(* CODESYS project verseny2

Project tree, tasks and I/O mapping:
  Device : CODESYS Control for PFC200 SL, 3S - Smart Software Solutions GmbH, version 4.1.0.0
    application Application
      libraries: Standard, * (System)
      task MainTask (cyclic, interval t#20ms, priority 1) calls MANUAL_TEST, input_led
      Andris/
        program prg_Beolvasas [ST]
        program prgBeolvasas_Sagaval_kezdunk [ST]
        program prgBeolvasas_Zoldel_kezdunk [ST]
      enum/
        data type enuIranyok
        data type enuMain
        data type enuSzinek
      data type enumRobotok
      fb/
        function block fbBLINKER2 [ST]
        function block fbBLINKER4 [ST]
        function block fbKombi3 [ST]
        function block fbKombi4 [ST]
      fun/
        function funAGV1_Location [ST]
        function funAGV2_Location [ST]
        function funAVG1_Set_Destination_1 [ST]
        function funAVG1_Set_Destination [ST]
        function funSargaElsoOszlopCheck [ST]
        function funTombfordito [ST]
        function funTombMaximuma [ST]
        function funTombMinimuma [ST]
        function funTombRendezesBuborek [ST]
        function funZoldElsoOszlopCheck [ST]
      global variables GVL
      global variables I
      program input_led [ST]
      Magocsi/
        function block fbMozgatas_zold [ST]
        function block fbRendezes [ST]
        function block fbRobotMozgas [ST]
      program MANUAL_TEST [ST]
      program PLC_PRG [ST]
      prg/
        program prgTEST1 [ST]
        program prgTEST2 [ST]
      global variables Q
      Ricsi/
        program prgEllenorzes [ST]
        program prgEmel [ST]
        program prgLerak [ST]
        program prgRaktar_sor1_bol_vegpontba [ST]
        program prgRaktarazas [ST]
        program prgSarga [ST]
        program prgZold [ST]
        program TEST [ST]
      program state_machine_main [ST]
    Pfc200Bus : Wago PFC200 internal bus, 3S - Smart Software Solutions GmbH, version 4.1.0.0
      _750_14xx : 16DI, WAGO Kontakttechnik GmbH u. Co. KG, order no. 750-14xx, version 4.1.0.0
          unmapped channels: %IW5 Digital Inputs 0 - 15
      _750_14xx_1 : 16DI, WAGO Kontakttechnik GmbH u. Co. KG, order no. 750-14xx, version 4.1.0.0
          unmapped channels: %IW20 Digital Inputs 0 - 15
      _750_15xx_1 : 16DO, WAGO Kontakttechnik GmbH u. Co. KG, order no. 750-15xx, version 4.1.0.0
          unmapped channels: %QW20 Digital Outputs 0 - 15
      _750_15xx : 16DO, WAGO Kontakttechnik GmbH u. Co. KG, order no. 750-15xx, version 4.1.0.0
          unmapped channels: %QW5 Digital Outputs 0 - 15
      _75x_459 : 75x-459/0..-000 4AI, 0-10 V, WAGO Kontakttechnik GmbH u. Co. KG, order no. 75x-459(/0..-000), version 4.1.0.0
          unmapped channels: Analog Input Channel 0, Analog Input Channel 1, Analog Input Channel 2, Analog Input Channel 3
      _75x_559 : 75x-559/0..-000 4AO, 0-10 V, WAGO Kontakttechnik GmbH u. Co. KG, order no. 75x-559(/0..-000), version 4.1.0.0
          unmapped channels: Analog Output Channel 0, Analog Output Channel 1, Analog Output Channel 2, Analog Output Channel 3
*)

// Device/Application/enumRobotok
{attribute 'qualified_only'}
{attribute 'strict'}
TYPE enumRobotok :
(
	AGV_Sarga,
	AGV_Zold
);
END_TYPE

// Device/Application/enum/enuIranyok
{attribute 'qualified_only'}
{attribute 'strict'}
TYPE enuIranyok :
(
	felfele,
	lefele,
	balra,
	jobbra
);
END_TYPE

// Device/Application/enum/enuMain
{attribute 'qualified_only'}
{attribute 'strict'}
TYPE enuMain :
(
	wait,
	init,
	beolvasas,
	rendezes,
	done
	
) := wait;
END_TYPE

// Device/Application/enum/enuSzinek
{attribute 'qualified_only'}
{attribute 'strict'}
TYPE enuSzinek :
(
	empty,
	zold,
	sarga,
	kek
);
END_TYPE

// Device/Application/GVL
{attribute 'qualified_only'}
VAR_GLOBAL
	start_r_trig: R_TRIG;
	start_f_trig: F_TRIG;
	stop_r_trig: R_TRIG;
	stop_f_trig: F_TRIG;
	emerg_r_trig: R_TRIG;
	emerg_f_trig: F_TRIG;
	
	aiTombSzinek: ARRAY [0..15] OF INT := [0,-1,-1,-1,-1,-1,-1,-1,-1,-1,0,0,0,0,0,0];
	axTombRobot1Zold: ARRAY [0..15] OF BOOL := [16(TRUE)];
	axTombRobot2Sarga: ARRAY [0..15] OF BOOL := [16(TRUE)];
END_VAR

// Device/Application/I
{attribute 'qualified_only'}
VAR_GLOBAL
	TEST0 AT %IX10.0 : BOOL;
	TEST1 AT %IX10.1 : BOOL;
	TEST2 AT %IX10.2 : BOOL;
	TEST3 AT %IX10.3 : BOOL;
	TEST4 AT %IX10.4 : BOOL;
	TEST5 AT %IX10.5 : BOOL;
	TEST6 AT %IX10.6 : BOOL;
	TEST7 AT %IX10.7 : BOOL;
	TEST8 AT %IX11.0 : BOOL;
	TEST9 AT %IX11.1 : BOOL;
	TEST10 AT %IX11.2 : BOOL;
	TEST11 AT %IX11.3 : BOOL;
	TEST12 AT %IX11.4 : BOOL;
	TEST13 AT %IX11.5 : BOOL;
	TEST14 AT %IX11.6 : BOOL;
	TEST15 AT %IX11.7 : BOOL;
	
	i0 AT %IX40.0 : BOOL;
	i1 AT %IX40.1 : BOOL;
	i2 AT %IX40.2 : BOOL;
	i3 AT %IX40.3 : BOOL;
	i4 AT %IX40.4 : BOOL;
	i5 AT %IX40.5 : BOOL;
	i6 AT %IX40.6 : BOOL;
	i7 AT %IX40.7 : BOOL;
	i8 AT %IX41.0 : BOOL;
	i9 AT %IX41.1 : BOOL;
	i10 AT %IX41.2 : BOOL;
	i11 AT %IX41.3 : BOOL;
	i12 AT %IX41.4 : BOOL;
	i13 AT %IX41.5 : BOOL;
	i14 AT %IX41.6 : BOOL;
	i15 AT %IX41.7 : BOOL;
END_VAR

// Device/Application/Q
{attribute 'qualified_only'}
VAR_GLOBAL
	TEST0 AT %QX10.0 : BOOL;
	TEST1 AT %QX10.1 : BOOL;
	TEST2 AT %QX10.2 : BOOL;
	TEST3 AT %QX10.3 : BOOL;
	TEST4 AT %QX10.4 : BOOL;
	TEST5 AT %QX10.5 : BOOL;
	TEST6 AT %QX10.6 : BOOL;
	TEST7 AT %QX10.7 : BOOL;
	TEST8 AT %QX11.0 : BOOL;
	TEST9 AT %QX11.1 : BOOL;
	TEST10 AT %QX11.2 : BOOL;
	TEST11 AT %QX11.3 : BOOL;
	TEST12 AT %QX11.4 : BOOL;
	TEST13 AT %QX11.5 : BOOL;
	TEST14 AT %QX11.6 : BOOL;
	TEST15 AT %QX11.7 : BOOL;
	
	q0 AT %QX40.0 : BOOL;
	q1 AT %QX40.1 : BOOL;
	q2 AT %QX40.2 : BOOL;
	q3 AT %QX40.3 : BOOL;
	q4 AT %QX40.4 : BOOL;
	q5 AT %QX40.5 : BOOL;
	q6 AT %QX40.6 : BOOL;
	q7 AT %QX40.7 : BOOL;
	q8 AT %QX41.0 : BOOL;
	q9 AT %QX41.1 : BOOL;
	q10 AT %QX41.2 : BOOL;
	q11 AT %QX41.3 : BOOL;
	q12 AT %QX41.4 : BOOL;
	q13 AT %QX41.5 : BOOL;
	q14 AT %QX41.6 : BOOL;
	q15 AT %QX41.7 : BOOL;
	

	
END_VAR

// Device/Application/MANUAL_TEST
PROGRAM MANUAL_TEST
VAR
END_VAR

//KONZOL MUKODTETI AZ OUTPUTOKAT
%QW20:= %IW5;

END_PROGRAM

// Device/Application/input_led
PROGRAM input_led
VAR
END_VAR

//INPUT A KONZOL LEDEKEN
%QW5:= %IW20;

END_PROGRAM

// Device/Application/PLC_PRG
PROGRAM PLC_PRG
VAR
END_VAR

END_PROGRAM

// Device/Application/state_machine_main
PROGRAM state_machine_main
VAR
	iState : enuMain;
	mem_robot : enumRobotok;
END_VAR

CASE iState OF
enuMain.wait:
	
	IF ( ( i.AGV1_L0 OR i.AGV1_L1 OR i.AGV1_L2 OR i.AGV1_L3 ) AND 
		(i.AGV2_L0 OR i.AGV2_L1 OR i.AGV2_L2 OR i.AGV2_L3)) THEN
		iState := enuMain.init;
	END_IF

enuMain.init:
	gvl.axTombRobot1Zold[funAGV1_Location()] := FALSE;
	gvl.axTombRobot2Sarga[funAGV2_Location()] := FALSE;
	IF gvl.axTombRobot1Zold[10] = FALSE THEN
		mem_robot := enumRobotok.AGV_Zold;
	ELSE
		mem_robot := enumRobotok.AGV_Sarga;
	END_IF
	
	iState := enuMain.beolvasas;	
enuMain.beolvasas:
	IF mem_robot = enumRobotok.AGV_Zold THEN
		prgBeolvasas_Zoldel_kezdunk();
	ELSE
		prgBeolvasas_Sagaval_kezdunk();
	END_IF
	
	IF prgBeolvasas_Sagaval_kezdunk.xDone OR prgBeolvasas_Zoldel_kezdunk.xDone THEN
		iState := enuMain.rendezes;
	END_IF 

	
enuMain.rendezes:
enuMain.done:	
END_CASE

END_PROGRAM

// Device/Application/fun/funAGV1_Location
FUNCTION funAGV1_Location : int
VAR_INPUT
END_VAR
VAR
END_VAR

funAGV1_Location := (TO_INT(i.AGV1_L0)) * 1 + (TO_INT(i.AGV1_L1)) * 2 
+ (TO_INT(i.AGV1_L2)) * 4 +(TO_INT( i.AGV1_L3)) * 8;
RETURN;

END_FUNCTION

// Device/Application/fun/funAGV2_Location
FUNCTION funAGV2_Location : int
VAR_INPUT
END_VAR
VAR
END_VAR

funAGV2_Location := i.AGV2_L0 * 1 + i.AGV2_L1 * 2 + i.AGV2_L2 * 4 + i.AGV2_L3 * 8;
RETURN;

END_FUNCTION

// Device/Application/Andris/prgBeolvasas_Zoldel_kezdunk
PROGRAM prgBeolvasas_Zoldel_kezdunk
VAR
	state_Zold : INT;
	state_Sarga : INT;
	lepesek_zold : INT;
	index1 : INT := 4;
	index2 : INT := 5;
	
	fbZold : fbRobotMozgas;
	fbSarga : fbRobotMozgas;
	
END_VAR

VAR_OUTPUT
	xDone : BOOL;
END_VAR

CASE state_Zold OF
// ZOLD MOZGATAS
0:
//10 - > 1
	fbZold(xEnable := TRUE , melyik_mozog := enumRobotok.AGV_Zold , merre_mozog := 1);
	IF fbZold.xDone THEN
		state_Zold := 1;
		gvl.aiTombSzinek[1] := TO_INT(i.AGV1_ID0)*1 + TO_INT(i.AGV1_ID1)*2;
	END_IF
1:
//1 - > 4 -> 7 -> 2
WHILE index1 > -1  DO
	fbZold(xEnable := TRUE , melyik_mozog := enumRobotok.AGV_Zold , merre_mozog := index1);
	
	IF fbZold.xDone THEN
	gvl.aiTombSzinek[index1] := TO_INT(i.AGV1_ID0)*1 + TO_INT(i.AGV1_ID1)*2;
		IF index1 = 7 THEN
			index1 := 8;	
		ELSE
			IF lepesek_zold <= 3 THEN
				index1 := index1 + 3;
			ELSE
				index1 := index1 - 3;
			END_IF
		END_IF
	lepesek_zold := lepesek_zold + 1;
	
	END_IF
	
END_WHILE

IF index1 < 0  THEN
	state_Zold := 3;
END_IF
3:
// DONE
END_CASE


CASE state_Sarga OF

0:
//15 -> 10
	fbSarga(xEnable := TRUE , merre_mozog := 10 , melyik_mozog := enumRobotok.AGV_Sarga );
	IF fbSarga.xDone THEN
		state_Sarga := 1;
	END_IF
1:
//10 -> 3	
	fbSarga(xEnable := TRUE , merre_mozog := 3 , melyik_mozog := enumRobotok.AGV_Sarga );
	IF fbSarga.xDone THEN
		state_Sarga := 2;
		gvl.aiTombSzinek[3] := TO_INT(i.AGV2_ID0)*1 + TO_INT(i.AGV2_ID1)*2;
	END_IF
2:
//3 -> 9
	WHILE index2 < 10  DO
		fbSarga(xEnable := TRUE , merre_mozog := index2 , melyik_mozog := enumRobotok.AGV_Sarga );
		IF fbSarga.xDone THEN
			gvl.aiTombSzinek[index2] := TO_INT(i.AGV2_ID0)*1 + TO_INT(i.AGV2_ID1)*2;
			index2 := index2 +3;
		END_IF

	END_WHILE
	
	IF index2 > 9 THEN
		state_Sarga := 3;
	END_IF
3:
//DONE
END_CASE

IF (state_Sarga = 3) AND (state_Zold = 3) THEN
	xDone := TRUE;
END_IF

END_PROGRAM

// Device/Application/Magocsi/fbRobotMozgas
FUNCTION_BLOCK fbRobotMozgas
VAR_INPUT
	melyik_mozog: INT;
	merre_mozog: INT;
	xEnable: BOOL;
END_VAR
VAR_OUTPUT
	xDone: BOOL;
END_VAR
VAR
	iStateRobotMozgas: INT;
END_VAR

IF NOT xEnable THEN
	RETURN;
END_IF

CASE melyik_mozog OF
	//zold robot
	enumRobotok.AGV_Zold:
		CASE iStateRobotMozgas OF
			0: 
				xDone := FALSE;
				
				funAVG1_Set_Destination(merre_mozog);
				q.AGV1_START := TRUE;
				
				iStateRobotMozgas := 1;
				
			1:
				IF funAGV1_Location() = 0 THEN
					q.AGV1_START := FALSE;
					
					iStateRobotMozgas := 2;
				END_IF
				
			2:
				IF funAgv1_location() > 0 THEN
					iStateRobotMozgas := 0;
					xDone := TRUE;
				END_IF
		END_CASE
		
	//sarga robot
	enumRobotok.AGV_Sarga:
		CASE iStateRobotMozgas OF
			0: 
				xDone := FALSE;
				
				funAVG2_Set_Destination(merre_mozog);
				q.AGV2_START := TRUE;
				
				iStateRobotMozgas := 1;
				
			1:
				IF funAGV2_Location() = 0 THEN
					q.AGV2_START := FALSE;
					
					iStateRobotMozgas := 2;
				END_IF
				
			2:
				IF funAgv2_location() > 0 THEN
					iStateRobotMozgas := 0;
					xDone := TRUE;
				END_IF
		END_CASE
END_CASE

END_FUNCTION_BLOCK

// Device/Application/fun/funAVG1_Set_Destination
FUNCTION funAVG1_Set_Destination : int
VAR_INPUT
	index : INT;
END_VAR
VAR
END_VAR

q.AGV1_D0 := index.0;
q.AGV1_D1 := index.1;
q.AGV1_D2 := index.2;
q.AGV1_D3 := index.3;

END_FUNCTION

// Device/Application/Andris/prgBeolvasas_Sagaval_kezdunk
PROGRAM prgBeolvasas_Sagaval_kezdunk
VAR
	state_Zold : INT;
	state_Sarga : INT;
	lepesek_zold : INT;
	lepesek_sarga : INT ;
	index1 : INT := 4;
	index2 : INT := 5;
	
	fbZold : fbRobotMozgas;
	fbSarga : fbRobotMozgas;
	
END_VAR

VAR_OUTPUT
	xDone : BOOL;
END_VAR

CASE state_Sarga OF
// Sarga MOZGATAS
0:
//10 - > 1
	fbSarga(xEnable := TRUE , melyik_mozog := enumRobotok.AGV_Sarga , merre_mozog := 1);
	IF fbSarga.xDone THEN
		state_Sarga := 1;
		gvl.aiTombSzinek[1] := TO_INT(i.AGV1_ID0)*1 + TO_INT(i.AGV1_ID1)*2;
	END_IF
1:
//1 - > 4 -> 7 -> 2
WHILE index1 > -1  DO
	fbSarga(xEnable := TRUE , melyik_mozog := enumRobotok.AGV_Sarga , merre_mozog := index1);
	
	IF fbSarga.xDone THEN
	gvl.aiTombSzinek[index1] := TO_INT(i.AGV1_ID0)*1 + TO_INT(i.AGV1_ID1)*2;
		IF index1 = 7 THEN
			index1 := 8;	
		ELSE
			IF lepesek_Sarga <= 3 THEN
				index1 := index1 + 3;
			ELSE
				index1 := index1 - 3;
			END_IF
		END_IF
	lepesek_Sarga := lepesek_Sarga + 1;
	
	END_IF
	
END_WHILE

IF index1 < 0  THEN
	state_Sarga := 3;
END_IF
3:
// DONE
END_CASE


CASE state_Zold OF

0:
//15 -> 10
	fbZold(xEnable := TRUE , merre_mozog := 10 , melyik_mozog := enumRobotok.AGV_Zold );
	IF fbZold.xDone THEN
		state_Zold := 1;
	END_IF
1:
//10 -> 3	
	fbZold(xEnable := TRUE , merre_mozog := 3 , melyik_mozog := enumRobotok.AGV_Zold );
	IF fbZold.xDone THEN
		state_Zold := 2;
		gvl.aiTombSzinek[3] := TO_INT(i.AGV2_ID0)*1 + TO_INT(i.AGV2_ID1)*2;
	END_IF
2:
//3 -> 9
	WHILE index2 < 10  DO
		fbZold(xEnable := TRUE , merre_mozog := index2 , melyik_mozog := enumRobotok.AGV_Zold );
		IF fbZold.xDone THEN
			gvl.aiTombSzinek[index2] := TO_INT(i.AGV2_ID0)*1 + TO_INT(i.AGV2_ID1)*2;
			index2 := index2 +3;
		END_IF

	END_WHILE
	
	IF index2 > 9 THEN
		state_Zold := 3;
	END_IF
3:
//DONE
END_CASE

IF (state_Sarga = 3) AND (state_Zold = 3) THEN
	xDone := TRUE;
END_IF

END_PROGRAM

// Device/Application/Andris/prg_Beolvasas
PROGRAM prg_Beolvasas
VAR
	state_Zold : INT;
	state_Sarga : INT;
	fbZold : fbRobotMozgas;
	fbSarga : fbRobotMozgas;
	index1 : INT := 4;
END_VAR

VAR_OUTPUT
	xDone : BOOL;
END_VAR

VAR_INPUT 
	Melyik_van_a_10_en : enumRobotok;
END_VAR

IF Melyik_van_a_10_en = enumRobotok.AGV_Zold THEN

CASE state_Zold OF
// ZOLD MOZGATAS
0:
//10 - > 1
	fbZold(xEnable := TRUE , melyik_mozog := enumRobotok.AGV_Zold , merre_mozog := 1);
	IF fbZold.xDone THEN
		state_Zold := 2;
	END_IF
2:
//1 - > 4 -> 7 -> 2
WHILE NOT (index1 = 2) DO
	
END_WHILE

3:
/

END_CASE

ELSE
	
END_IF

END_PROGRAM

// Device/Application/fb/fbBLINKER2
(*
EZ A FUNKCIO BLOK EGY VILLOGOT VALOSIT MEG AMINEK MINT 
A BEKAPCSOLT IDEJÉT MINT A KIKAPCSOLT IDEJÉT TUDJUK ÁLLITANI.
*)
FUNCTION_BLOCK fbBLINKER2 
VAR_INPUT
	ENABLE : BOOL;
	TIME_ON : TIME ;
	TIME_OFF : TIME;
END_VAR
VAR_OUTPUT
	Q : BOOL;
END_VAR
VAR
	TIMER1 : TON;
	TIMER2 : TON;
	state : INT := 0;
END_VAR

IF ENABLE THEN

TIMER1(IN := state = 0,PT := TIME_ON);
TIMER2(IN := state = 1  , PT := TIME_OFF);

CASE state OF
0:
// ON 
	Q := TRUE;
	IF timer1.Q THEN
		state := 1;
	END_IF
1:
// OFF
	Q := FALSE;
	IF timer2.Q THEN
		state := 0;
	END_IF
	
END_CASE
ELSE
	q := false;
END_IF

END_FUNCTION_BLOCK

// Device/Application/fb/fbBLINKER4
(*
EZ A FUNKCIO BLOK EGY DUPLA VILLOGOT VALOSIT MEG AMINEK MINT 
A BEKAPCSOLT IDEJÉT MINT A KIKAPCSOLT IDEJÉT TUDJUK ÁLLITANI.
*)
FUNCTION_BLOCK fbBLINKER4 
VAR_INPUT
	ENABLE : BOOL;
	TIME_ON1 : TIME ;
	TIME_OFF1 : TIME;
	TIME_ON2 : TIME ;
	TIME_OFF2 : TIME;
END_VAR
VAR_OUTPUT
	Q : BOOL;
END_VAR
VAR
	TIMER0 : TON;
	TIMER1 : TON;
	TIMER2 : TON;
	TIMER3 : TON;
	state : INT := 0;
END_VAR

IF ENABLE THEN

TIMER0(IN := state = 0  , PT := TIME_ON1);
TIMER1(IN := state = 1  , PT := TIME_OFF1);
TIMER2(IN := state = 2  , PT := TIME_ON2);
TIMER3(IN := state = 3  , PT := TIME_OFF2);

CASE state OF
0:
// ON1
	Q := TRUE;
	IF timer0.Q THEN
		state := 1;
	END_IF
1:
// OFF1
	Q := FALSE;
	IF timer1.Q THEN
		state := 2;
	END_IF
2:
// ON2
	Q := TRUE;
	IF timer2.Q THEN
		state := 3;
	END_IF
3:
// OFF2
	Q := FALSE;
	IF timer3.Q THEN
		state := 0;
	END_IF
	
END_CASE
ELSE
	q := FALSE ;
END_IF

END_FUNCTION_BLOCK

// Device/Application/fb/fbKombi3
(*
EZ A FUNKCIO BLOK EGY 3 BEMENETÜ KOMBINÁCIOS HÁLLOZATOT VALOSIT MEG.
A HÁLLOZAT IGAZSÁG TÁBLÁJÁT TÁROLJA
*)
FUNCTION_BLOCK fbKombi3
VAR
	index : INT;
END_VAR
VAR_INPUT
	A : BOOL; // NULLADIK HELYIÉRTÉK
	B : BOOL; // ELSÖ HELYIÉRTÉK
	C : BOOL; // MÁSODIK HELYIÉRTÉK
	TABLE : ARRAY[0..7] OF BOOL; // IGAZSÁG TÁBLA A ELEM INDEXE MEGEGYEZIK A MINTERM SZÁMMAL
END_VAR
VAR_OUTPUT
	Q : BOOL ; // KIMENET
END_VAR

index := 1*TO_INT(A) + 2*TO_INT(B) + 4*TO_INT(C);
Q := TABLE[index];

END_FUNCTION_BLOCK

// Device/Application/fb/fbKombi4
(*
EZ A FUNKCIO BLOK EGY 3 BEMENETÜ KOMBINÁCIOS HÁLLOZATOT VALOSIT MEG.
A HÁLLOZAT IGAZSÁG TÁBLÁJÁT TÁROLJA
*)
FUNCTION_BLOCK fbKombi4
VAR
	index : INT;
END_VAR
VAR_INPUT
	A : BOOL; // NULLADIK HELYIÉRTÉK
	B : BOOL; // ELSÖ HELYIÉRTÉK
	C : BOOL; // MÁSODIK HELYIÉRTÉK
	D : BOOL; // HARMADIK HELYIÉRTÉK
	TABLE : ARRAY[0..15] OF BOOL; // IGAZSÁG TÁBLA A ELEM INDEXE MEGEGYEZIK A MINTERM SZÁMMAL
END_VAR
VAR_OUTPUT
	Q : BOOL ; // KIMENET
END_VAR

index := 1*TO_INT(A) + 2*TO_INT(B) + 4*TO_INT(C) + 4*TO_INT(D); 
Q := TABLE[index];

END_FUNCTION_BLOCK

// Device/Application/fun/funAVG1_Set_Destination_1
FUNCTION funAVG1_Set_Destination_1 : int
VAR_INPUT
	index : int;
END_VAR
VAR
END_VAR

q.AGV2_D0 := index.0;
q.AGV2_D1 := index.1;
q.AGV2_D2 := index.2;
q.AGV2_D3 := index.3;

END_FUNCTION

// Device/Application/fun/funSargaElsoOszlopCheck
FUNCTION funSargaElsoOszlopCheck : INT;
VAR_INPUT
END_VAR
VAR
	iIndex : INT;
END_VAR

WHILE (GVL.aiTombSzinek[iindex] <> enuszinek.sarga) DO
	iIndex := iindex + 1;
END_WHILE

funSargaElsoOszlopCheck := iindex;

END_FUNCTION

// Device/Application/fun/funTombfordito
FUNCTION funTombfordito
VAR_IN_OUT
	aiTomb: ARRAY [*] OF INT;
END_VAR
VAR
	iTemp: INT;
	iIndex: DINT;
	iFelso: DINT := UPPER_BOUND(aiTomb, 1);
	iKozep: DINT := ((UPPER_BOUND(aiTomb, 1) - LOWER_BOUND(aiTomb, 1)) / 2);
END_VAR

FOR iIndex := LOWER_BOUND(aiTomb, 1) TO iKozep DO
	iTemp := aiTomb[iIndex];
	aiTomb[iIndex] := aiTomb[iFelso - iIndex];
	aiTomb[iFelso - iIndex] := iTemp;
END_FOR

END_FUNCTION

// Device/Application/fun/funTombMaximuma
FUNCTION funTombMaximuma : INT
VAR_IN_OUT
	aiTomb: ARRAY [*] OF INT;
END_VAR
VAR
	iIndexLegnagyobb: DINT := LOWER_BOUND(aiTomb, 1);
	iIndexJelenlegVizsgalt: DINT;
END_VAR
VAR_INPUT
	xElsotAdjaVissza: BOOL;
END_VAR

FOR iIndexJelenlegVizsgalt := iIndexLegnagyobb + 1 TO UPPER_BOUND(aiTomb, 1) DO
	IF (xElsotAdjaVissza AND (aiTomb[iIndexJelenlegVizsgalt] > aiTomb[iIndexLegnagyobb])) OR (NOT xElsotAdjaVissza AND (aiTomb[iIndexJelenlegVizsgalt] >= aiTomb[iIndexLegnagyobb])) THEN
		iIndexLegnagyobb := iIndexJelenlegVizsgalt;
	END_IF
END_FOR

funTombMaximuma := TO_INT(iIndexLegnagyobb);

END_FUNCTION

// Device/Application/fun/funTombMinimuma
FUNCTION funTombMinimuma : INT
VAR_IN_OUT
	aiTomb: ARRAY [*] OF INT;
END_VAR
VAR
	iIndexLegkisebb: DINT := LOWER_BOUND(aiTomb, 1);
	iIndexJelenlegVizsgalt: DINT;
END_VAR
VAR_INPUT
	xElsotAdjaVissza: BOOL;
END_VAR

FOR iIndexJelenlegVizsgalt := iIndexLegkisebb + 1 TO UPPER_BOUND(aiTomb, 1) DO
	IF (xElsotAdjaVissza AND (aiTomb[iIndexJelenlegVizsgalt] < aiTomb[iIndexLegkisebb])) OR (NOT xElsotAdjaVissza AND (aiTomb[iIndexJelenlegVizsgalt] <= aiTomb[iIndexLegkisebb])) THEN
		iIndexLegkisebb := iIndexJelenlegVizsgalt;
	END_IF
END_FOR

funTombMinimuma := TO_INT(iIndexLegkisebb);

END_FUNCTION

// Device/Application/fun/funTombRendezesBuborek
FUNCTION funTombRendezesBuborek
VAR_IN_OUT
	aiTomb: ARRAY [*] OF INT;
END_VAR
VAR
	iElsoIndex: DINT := LOWER_BOUND(aiTomb, 1);
	iUtolsoIndex: DINT := UPPER_BOUND(aiTomb, 1);
	iIndexBelso: DINT;
	iIndexKulso: DINT;
	iTemp: INT;
END_VAR
VAR_INPUT
END_VAR

FOR iIndexKulso := iElsoIndex TO iUtolsoIndex - 1 DO
	FOR iIndexBelso := iElsoIndex TO (iUtolsoIndex - iIndexKulso - 1) DO
		IF aiTomb[iIndexBelso] > aiTomb[iIndexBelso + 1] THEN
			iTemp := aiTomb[iIndexBelso];
			aiTomb[iIndexBelso] := aiTomb[iIndexBelso + 1];
			aiTomb[iIndexBelso + 1] := iTemp;
		END_IF
	END_FOR
END_FOR

END_FUNCTION

// Device/Application/fun/funZoldElsoOszlopCheck
FUNCTION funZoldElsoOszlopCheck : INT;
VAR_INPUT
END_VAR
VAR
	iIndex : INT;
END_VAR

WHILE (GVL.aiTombSzinek[iindex] <> enuszinek.zold) DO
	iIndex := iIndex + 1;
END_WHILE

funZoldElsoOszlopCheck := iindex;

END_FUNCTION

// Device/Application/Magocsi/fbMozgatas_zold
FUNCTION_BLOCK fbMozgatas_zold
VAR_INPUT
	hova: INT;
END_VAR
VAR_OUTPUT
	xdone: BOOL;
END_VAR
VAR
	istate : INT;
	ifuggoleges: INT;
	ivizszintes: INT;
	fbrobotmozgas :fbrobotmozgas;
END_VAR

CASE istate OF
	0:
		xdone := FALSE;
		IF funAGV1_Location() -3 > 0 THEN
			ifuggoleges := ifuggoleges + 1;
		END_IF
		
		IF funAGV1_Location() -3 > 0 THEN
			ifuggoleges := ifuggoleges + 1;
		END_IF
		
		IF funAGV1_Location() -1 > 0 THEN
			ivizszintes := ivizszintes + 1;
		END_IF
		
		IF funagv1_location() - 1 > 0 THEN
			ivizszintes := ivizszintes + 1;
		END_IF
		
		istate := 1;
	1:
		fbrobotmozgas(melyik_mozog:= enumRobotok.AGV_zold, merre_mozog:= ivizszintes * 3 + funAGV1_Location() - ifuggoleges, xEnable:= TRUE);
		
		IF fbrobotmozgas.xDone THEN
			ifuggoleges := ifuggoleges - 1;
			
		END_IF
		
		IF ifuggoleges = 0 THEN
			istate := 2;
		END_IF
		
	2:
		fbrobotmozgas(melyik_mozog:= enumRobotok.AGV_Zold, merre_mozog:= funagv1_location() - (ivizszintes *3), xenable := TRUE);
		
		IF fbrobotmozgas.xDone THEN
			ivizszintes := ivizszintes - 1;
		END_IF
		
		IF ivizszintes = 0 THEN
			xdone := TRUE;
			istate := 0;
		END_IF
END_CASE

END_FUNCTION_BLOCK

// Device/Application/Magocsi/fbRendezes
FUNCTION_BLOCK fbRendezes
VAR_INPUT
END_VAR
VAR_OUTPUT
	xdone : BOOL;
END_VAR
VAR
	iIndexElsoSzines : INT;
	iindexelsolyuk: INT;
	istate: INT;
	aikicsi: ARRAY [0..5] OF INT := [5,8,7,4,1,2];
	ainagy: ARRAY [0..8] OF INT := [6,9,8,7,4,1,2,3];
	kulonbseg: INT;
	iai: INT;
	fbrobotmozgas: fbrobotmozgas;
	fbMozgatas_zold: fbMozgatas_zold;
END_VAR

CASE istate OF
	0:
	iai := 0;
	iindexelsoszines := 0;
	iindexelsolyuk := 0;
	xDone := FALSE;
	
	WHILE (GVL.aiTombSzinek[iIndexElsoSzines] <> enuszinek.zold) OR (GVL.aiTombSzinek[iindexelsoszines] <> enuszinek.sarga) DO
	iindexelsoszines := iIndexElsoSzines + 1;
END_WHILE

WHILE GVL.aiTombSzinek[iindexelsolyuk] <> enuszinek.empty DO
	iindexelsolyuk := iindexelsolyuk + 1;
END_WHILE

kulonbseg := (iindexelsolyuk MOD 3) - (iIndexElsoSzines MOD 3);

	 IF (kulonbseg >= -1) AND (kulonbseg <=1) THEN
		iState := 1;
		WHILE aikicsi[iai] <> iindexelsolyuk DO
			iai := iai + 1;
		END_WHILE
	 ELSE
		 iState := 5;
		 WHILE ainagy[iai] <> iindexelsolyuk DO
			iai := iai + 1;
		END_WHILE
	 END_IF
	 
	1:
		fbmozgatas_zold;
		IF fbMozgatas_zold.xdone THEN
			istate := 2;
		END_IF
	2:
		IF (funSargaElsoOszlopCheck() > 0) THEN
			istate := 8;
		ELSIF (funZoldElsoOszlopCheck() > 0) THEN
			xDone := TRUE;
			istate := 0;
			RETURN;
		END_IF
		
		prgEmel(melyik_emel:= enumRobotok.AGV_Zold);
		
		IF prgEmel.xDone THEN
			istate := 3;
		END_IF
		
	3:
		fbrobotmozgas(melyik_mozog:= enumrobotok.agv_zold, merre_mozog:= aikicsi[iai], xEnable:= TRUE);
		
		IF fbrobotmozgas.xDone THEN
			istate := 4;
		END_IF
		
	4:
		prgLerak(melyik_lerak:= enumrobotok.AGV_Zold);
		
		IF prgLerak.xDone THEN
			iai := iai + 1;
			
			IF iai = 6 THEN
				iai := 0;
			END_IF
		
			istate := 2;
		END_IF
		
	5:
		IF (funSargaElsoOszlopCheck() > 0) OR (funZoldElsoOszlopCheck() > 0) THEN
			xDone := TRUE;
			istate := 0;
			RETURN;
		END_IF
		
		prgEmel(melyik_emel:= enumRobotok.AGV_Zold);
		
		IF prgEmel.xDone THEN
			istate := 6;
		END_IF
		
	6:
		fbrobotmozgas(melyik_mozog:= enumrobotok.agv_zold, merre_mozog:= ainagy[iai], xEnable:= TRUE);
		
		IF fbrobotmozgas.xDone THEN
			istate := 7;
		END_IF
		
	7: 
	prgLerak(melyik_lerak:= enumrobotok.AGV_Zold);
		
		IF prgLerak.xDone THEN
			iai := iai + 1;
			
			IF iai = 8 THEN
				iai := 0;
			END_IF
		
			istate := 5;
		END_IF
	8:
		fbMozgatas_zold;
		fbrobotmozgas(melyik_mozog:= enumRobotok.AGV_Sarga, merre_mozog:= funSargaElsoOszlopCheck, xEnable:= TRUE);
END_CASE

END_FUNCTION_BLOCK

// Device/Application/Ricsi/prgEmel
PROGRAM prgEmel
VAR
	state : INT;
	robot1_emel :BOOL;
	robot2_emel :BOOL;
END_VAR
VAR_INPUT
	melyik_emel : INT;
END_VAR
VAR_OUTPUT
	xDone :BOOL;
END_VAR

//STATE
CASE STATE OF
0: //emel
	xDone := FALSE;
	IF melyik_emel = enumRobotok.AGV_Zold THEN
		q.AGV1_Pickup := TRUE;
		q.AGV2_Pickup := FALSE;
		robot1_emel := TRUE;
	END_IF
	IF melyik_emel = enumRobotok.AGV_Sarga THEN
		q.AGV1_Pickup := FALSE;
		q.AGV2_Pickup := TRUE;
		robot2_emel := TRUE;
	END_IF

1: // stop
	xDone := TRUE;
	IF melyik_emel = enumRobotok.AGV_Zold THEN
		q.AGV1_Pickup := FALSE;
	END_IF
	IF melyik_emel = enumRobotok.AGV_Sarga THEN
		q.AGV2_Pickup := FALSE;
	END_IF
END_CASE


//TRANSITION
CASE STATE OF
0: //emel
	IF robot1_emel AND i.AGV1_UP THEN
		state := 1;
	END_IF
	IF robot2_emel AND i.AGV2_DOWN THEN
		state := 1;
	END_IF
	
1: //stop

END_CASE

END_PROGRAM

// Device/Application/Ricsi/prgLerak
PROGRAM prgLerak
VAR
	state : INT := 0;
	robot1_le :BOOL := 0;
	robot2_le :BOOL := 0;
END_VAR
VAR_INPUT
	melyik_lerak : INT;
END_VAR
VAR_OUTPUT
	xDone :BOOL := 0;
END_VAR

//STATE
CASE state OF
0: //lerak
	xDone := FALSE;
	IF melyik_lerak = enumRobotok.AGV_Zold THEN
		q.AGV1_Drop := TRUE;
// 		q.AGV2_Drop := FALSE;
		robot1_le := TRUE;
	END_IF
	IF melyik_lerak = enumRobotok.AGV_Sarga THEN
// 		q.AGV1_Drop := FALSE;
		q.AGV2_Drop := TRUE;
		robot2_le := TRUE;
	END_IF
1: //stop
	IF melyik_lerak = enumRobotok.AGV_Zold THEN
		q.AGV1_Drop := FALSE;
		robot1_le := FALSE;
	END_IF
	IF melyik_lerak = enumRobotok.AGV_Sarga THEN
		q.AGV2_Drop := FALSE;
		robot2_le := FALSE;
	END_IF
	xDone := TRUE;
	state := 0;
END_CASE

//TRANSITION
CASE STATE OF
0: //lerak
	IF robot1_le AND i.AGV1_DOWN THEN
		state := 1;
	END_IF
	IF robot2_le AND i.AGV2_DOWN THEN
		state := 1;
	END_IF
	
END_CASE

END_PROGRAM

// Device/Application/prg/prgTEST1
PROGRAM prgTEST1
VAR
END_VAR

END_PROGRAM

// Device/Application/prg/prgTEST2
PROGRAM prgTEST2
VAR
	fbMozgat  : fbRobotMozgas;
END_VAR

IF %IX10.1 THEN
IF %IX10.0 THEN
	fbMozgat(xEnable := TRUE , melyik_mozog := enumRobotok.AGV_Sarga , merre_mozog := 1);
	ELSE
	fbMozgat(xEnable := TRUE , melyik_mozog := enumRobotok.AGV_Zold , merre_mozog := 1);
END_IF
END_IF

END_PROGRAM

// Device/Application/Ricsi/prgEllenorzes
PROGRAM prgEllenorzes
VAR
	state :INT := 0;
	ROBOT : fbRobotMozgas;
END_VAR
VAR_OUTPUT
	xDone :BOOL;
END_VAR

CASE state OF
0: //mozgat 15-be
	xDone := FALSE;
	ROBOT(melyik_mozog:= enumRobotok.AGV_Sarga, merre_mozog:= 15, xEnable:= TRUE);
1: //operator hivas
	Q.AGV2_OPERATOR := TRUE;
2: //operator hivas vege
	Q.AGV2_OPERATOR := FALSE;
	
END_CASE

CASE state OF
0:
	IF ROBOT.xDone THEN
		STATE := 1;
	END_IF
1:
	IF
		NOT I.AGV1_L0 AND NOT I.AGV1_L1 AND
		NOT I.AGV1_L2 AND NOT I.AGV1_L3 THEN
			state := 2;
	END_IF
2:
	IF 
		I.AGV1_L0 AND I.AGV1_L1 AND
		I.AGV1_L2 AND I.AGV1_L3 THEN
			state := 0;
			xDone := TRUE;
	END_IF
END_CASE

END_PROGRAM

// Device/Application/Ricsi/prgRaktar_sor1_bol_vegpontba
PROGRAM prgRaktar_sor1_bol_vegpontba
VAR
	zold :BOOL;
	sarga : BOOL;
	mozog : fbRobotMozgas
END_VAR

VAR_INPUT
	state :INT := 0;
END_VAR

VAR_OUTPUT
	xdone : BOOL;
END_VAR

CASE state OF
0: //tufunk semmit
	IF funZoldElsoOszlopCheck() > 0 THEN
		state := 1;
	ELSIF funSargaElsoOszlopCheck() > 0 THEN
		state := 2;
	END_IF
1:
prgZold(); //tufunk zold
	IF prgZold.xdone THEN
		state := 0;
		xdone := FALSE;
	END_IF
2:
prgSarga();
	IF prgSarga THEN
		state := 0;
		xdone := FALSE;
	END_IF
END_CASE




// CASE state OF 
// 0: // szin check
// 	zold := FALSE;
// 	sarga := FALSE;
// 	IF funZoldElsoOszlopCheck() > 0 THEN
// 		zold := TRUE;
// 		mozog(melyik_mozog:= enumRobotok.AGV_Zold, merre_mozog:= 10, xEnable:= TRUE);
// 	ELSIF funSargaElsoOszlopCheck() > 0 THEN
// 		sarga := TRUE;
// 		mozog(melyik_mozog:= enumRobotok.AGV_Sarga, merre_mozog:= 10, xEnable:= TRUE);
// 	END_IF
// 1: //
// END_CASE
// 
// 
// CASE state OF 
// 	
// END_CASE

END_PROGRAM

// Device/Application/Ricsi/prgZold
PROGRAM prgZold
VAR
	state : INT := 0;
	fbRobotMozgas : fbRobotMozgas;
END_VAR
VAR_OUTPUT
	xdone : BOOL := 0;
END_VAR

CASE state OF 
0: //mozgat 10 be
	xdone := FALSE;
	fbRobotMozgas(melyik_mozog:= enumRobotok.AGV_Zold, merre_mozog:= 10, xEnable:= TRUE);	
1: //raktarazas
	prgRaktarazas(melyik_robot:= enumRobotok.AGV_Zold);
END_CASE


CASE state OF 
0: //mozgat 10 be
	IF fbRobotMozgas.xDone THEN
		state := 1;
	END_IF
1: //raktarazas
	IF prgRaktarazas.xdone THEN
		xdone := FALSE;
		state := 0;
	END_IF
END_CASE

END_PROGRAM

// Device/Application/Ricsi/prgRaktarazas
PROGRAM prgRaktarazas
VAR
	xdone : BOOL;
	state : INT := 0;
	zold_hely_11 :BOOL := FALSE;
	zold_hely_12 :BOOL := FALSE;
	
	sarga_hely_13 :BOOL := FALSE;
	sarga_hely_14 :BOOL := FALSE;
	mozgat : fbRobotMozgas;
END_VAR

VAR_INPUT
	melyik_robot : INT;
END_VAR

// VAR_OUTPUT
// 	hova_rakta_le :INT;
// END_VAR

//ACTION
CASE state OF
0: //mozgatas
	IF melyik_robot := enumRobotok.AGV_Zold THEN
		IF zold_hely_12 = FALSE THEN
			mozgat(melyik_mozog:= enumRobotok.AGV_Zold, merre_mozog:= 12, xEnable:= TRUE);
		ELSIF zold_hely_11 = FALSE THEN
 			mozgat(melyik_mozog:= enumRobotok.AGV_Zold, merre_mozog:= 11, xEnable:= TRUE);
		END_IF
	ELSIF melyik_robot := enumRobotok.AGV_Sarga THEN
		IF sarga_hely_14 = FALSE THEN
			mozgat(melyik_mozog:= enumRobotok.AGV_Sarga, merre_mozog:= 14, xEnable:= TRUE);
		ELSIF sarga_hely_13 = FALSE THEN
 			mozgat(melyik_mozog:= enumRobotok.AGV_Sarga, merre_mozog:= 13, xEnable:= TRUE);
		END_IF
	END_IF
1: //lerakas
	IF melyik_robot := enumRobotok.AGV_Zold THEN
		prgLerak(melyik_lerak:= enumRobotok.AGV_Zold);
	ELSIF melyik_robot := enumRobotok.AGV_Sarga THEN
		prgLerak(melyik_lerak:= enumRobotok.AGV_Sarga);
	END_IF
2: //vissza 10-be
	IF melyik_robot := enumRobotok.AGV_Zold THEN
		mozgat(melyik_mozog:= enumRobotok.AGV_Zold, merre_mozog:= 10, xEnable:= TRUE);
	ELSIF melyik_robot := enumRobotok.AGV_Sarga THEN
		mozgat(melyik_mozog:= enumRobotok.AGV_Sarga, merre_mozog:= 10, xEnable:= TRUE);
	END_IF
END_CASE

//TRANSITION
CASE state OF
0:
	IF mozgat.xDone THEN
		state := 1;
	END_IF
1:
	IF prgLerak.xDone THEN
		state := 2;
	END_IF
2:
	IF mozgat.xDone THEN
		state := 0;
		xdone := 0;
	END_IF
END_CASE

END_PROGRAM

// Device/Application/Ricsi/prgSarga
PROGRAM prgSarga
VAR
	state : INT := 0;
	fbRobotMozgas : fbRobotMozgas;
END_VAR
VAR_OUTPUT
	xdone : BOOL := 0;
END_VAR

CASE state OF 
0: //mozgat 10 be
	xdone := FALSE;
	fbRobotMozgas(melyik_mozog:= enumRobotok.AGV_Sarga, merre_mozog:= 10, xEnable:= TRUE);
1: //ellenorgzes
	prgEllenorzes();
2: //raktarazas
	prgRaktarazas(melyik_robot:= enumRobotok.AGV_Sarga);
3: // 10-be
	fbRobotMozgas(melyik_mozog:= enumRobotok.AGV_Sarga, merre_mozog:= 10, xEnable:= TRUE);
// 4: // 2-be
// 	fbRobotMozgas(melyik_mozog:= enumRobotok.AGV_Sarga, merre_mozog:= 2, xEnable:= TRUE);
END_CASE


CASE state OF 
0: //mozgat 10 be
	IF fbRobotMozgas.xDone THEN
		state := 1;
	END_IF
1: //ellenorgzes
	IF prgEllenorzes.xDone THEN
		state := 2;
	END_IF
2: //raktarazas
	IF prgRaktarazas.xdone THEN
		state := 3;
	END_IF
3: //10be
	IF fbRobotMozgas.xDone THEN
		state := 0;
		xdone := TRUE;
	END_IF
// 4:
// 	IF fbRobotMozgas.xDone THEN
// 		xdone := TRUE;
// 		state := 0;
// 	END_IF
END_CASE

END_PROGRAM

// Device/Application/Ricsi/TEST
PROGRAM TEST
VAR
	state : INT;
	i :int;
END_VAR

CASE state OF
	0:
	prgEmel(melyik_emel:= enumRobotok.AGV_Zold);
	1:
	prgLerak(melyik_lerak:= enumRobotok.AGV_Zold);
	2:
	prgEllenorzes();
	3:
	prgRaktarazas(melyik_robot:= enumRobotok.AGV_Zold);
69:
	i := 69;
END_CASE


CASE state OF
	0:
	IF prgEmel.xDone THEN
		state := state + 1;
	END_IF
	1:
	IF prgLerak.xDone THEN
		state := state + 1;
	END_IF
	2:
	IF prgEllenorzes.xDone THEN
		state := state + 1;
	END_IF
	3:
	IF prgRaktarazas.xdone THEN
		state := 69;
	END_IF
END_CASE

END_PROGRAM
